INTERFACE I_CalculateHFromAngle


METHOD CalculateH : LREAL
VAR_INPUT
    Radians : LREAL;
END_VAR
VAR_OUTPUT
    Error : BOOL;
    ErrorMsg : T_MaxString;
END_VAR
END_METHOD


METHOD CalculateHVelocity : LREAL
VAR_INPUT
    Radians : LREAL;
    RadiansPerSecond : LREAL;
END_VAR
VAR_OUTPUT
    Error : BOOL;
    ErrorMsg : T_MaxString;
END_VAR
END_METHOD

END_INTERFACE

(* stored: Version 1.1.0.1, ProductVersion 3.1.4026.11
   Itf I_CalculateHFromAngle: Id {328e0bc5-0aab-4a8e-bb2c-40536669a0df}
   Method CalculateH: Id {e35eba4d-1f64-49b6-8bd4-c71c66f68688}
   Method CalculateHVelocity: Id {d309911d-27d4-4e4d-b3a1-8943968a718b} *)
